// TwinCAT 3 PLC project Display_100
// ProgramVersion: 3.1.4024.0
// libraries:
//   Tc2_Standard, * (Beckhoff Automation GmbH)
//   Tc2_System, * (Beckhoff Automation GmbH)
//   Tc3_Module, * (Beckhoff Automation GmbH)
// project tree:
//   / PlcTask.TcTTO
//   POUs/ MAIN.TcPOU
// (motion and I/O tree: see PLC project potentiometer_inlezen)
// real-time tasks:
//   TASK PlcTask: cycle T#10ms, priority 20, ADS port 350
//   TASK PlcTask1: cycle T#10ms, priority 21, ADS port 351
//   TASK PlcTask2: cycle T#10ms, priority 22, ADS port 352
//   TASK PlcTask3: cycle T#10ms, priority 26, ADS port 353
//   TASK PlcTask4: cycle T#10ms, priority 25, ADS port 354
//   TASK PlcTask5: cycle T#10ms, priority 24, ADS port 355
//   TASK PlcTask6: cycle T#10ms, priority 23, ADS port 356
//   TASK PlcTask7: cycle T#10ms, priority 27, ADS port 357

CONFIGURATION Display_100
    RESOURCE PLC ON TwinCAT3
        TASK PlcTask(INTERVAL := T#10ms, PRIORITY := 24);
        PROGRAM MAIN WITH PlcTask : MAIN;
    END_RESOURCE
END_CONFIGURATION

// ---- POUs/MAIN.TcPOU
PROGRAM MAIN
VAR

    fPotmeter: REAL; // De gemeten waarde van de potentiometer (0 tot 32767)
    displayValue: INT; // De waarde om weer te geven op het display (-100 tot +2000)


END_VAR

(*
Display_100 (2 regels)

Toon het voltage dat over de potentiometer staat op het display. Dit is een spanning met een maximale spanning van 10v, tevens de maximum inleesbare spanning van de EL3062 kaart die we gebruiken.

Opmerking: het fysieke display dat wij gebruiken is ingesteld om de waarden van -100 tot +2.000 weer te geven voor de respectievelijk 0v tot 10v spanning die het binnenkrijgt.
*)

// Omrekenen van de gemeten waarde naar de display waarde
displayValue := TO_INT((fPotmeter / 32767.0) * (2000 - (-100)) + (-100));

END_PROGRAM
